ABB RAPID module: Module2.modx

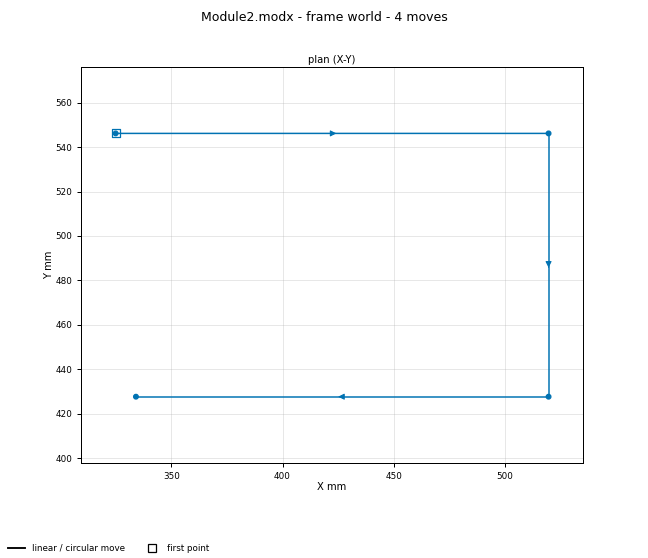
[picture p0: tool path of Module2.modx in frame world, 4 of 4 moves have a stored position in this frame; points joined in program order, loops and branches not executed]
MODULE Module2

    PROC Pohyb_po_drahe()
        MoveL [[324.881711325,546.154233124,230],[0.071763508,-0.988676922,-0.017208217,-0.130659179],[0,-1,2,0],[9E+09,9E+09,9E+09,9E+09,9E+09,9E+09]],v100,z10,tool0\WObj:=wobj0;
        MoveL [[519.705421258,546.154312597,230],[0.071763494,-0.988676918,-0.017208304,-0.1306592],[0,-1,2,0],[9E+09,9E+09,9E+09,9E+09,9E+09,9E+09]],v100,z10,tool0\WObj:=wobj0;
        MoveL [[519.705411147,427.668300637,230],[0.071763501,-0.988676918,-0.017208293,-0.1306592],[0,-1,2,0],[9E+09,9E+09,9E+09,9E+09,9E+09,9E+09]],v100,z10,tool0\WObj:=wobj0;
        MoveL [[334.023715996,427.668295879,230],[0.071763488,-0.98867692,-0.017208299,-0.130659188],[0,-1,2,0],[9E+09,9E+09,9E+09,9E+09,9E+09,9E+09]],v100,z10,tool0\WObj:=wobj0;
    ENDPROC

ENDMODULE
